INTERFACE INTERNAL I_ReceiverNode EXTENDS Debug.I_Debug

PROPERTY INTERNAL IsOk : BOOL
GET
END_GET
END_PROPERTY

METHOD INTERNAL Receive
VAR_INPUT
	iArg			: I_Arg;
END_VAR
END_METHOD

END_INTERFACE

(* stored: Version 1.1.0.1
   Itf I_ReceiverNode: Id {a66ea0f3-4a91-4fa0-8d6e-872222a657a8}
   Property IsOk: Id {21845255-3d04-4d9a-a4c8-4a3125bc4b09}
   Get Get: Id {70d0de8f-d4a9-4c14-9aa4-7ebd6f9e97be}
   Method Receive: Id {0ad5f0f9-72c2-4773-920a-c7c616371a13} *)
